Staubli VAL3: TrajJoint.pjx

--- TrajJoint.pjx ---
Parameters version=s7.2.1 stackSize=5000 millimeterUnit=true
Data file=TrajJoint.dtx
Type name=TrajJointItem path=Disk://kernel/template/TrajJointItem/TrajJointItem.pjx

--- TrajJoint.dtx ---
public num nIndexTool
public TrajJointItem tData
  [0]
    jointRx jJoint
    TrajectoryItem tSuper
      [0]
        num distance
        num moveType
        num nTime
        num nStop
        num nTcpAction
        string comment
        bool toStop
        mdesc nom_speed = {tmax=9999}
        InstrItem iInstr[3]
          [0]
            string sType
            string sData
          [1]
            string sType
            string sData
          [2]
            string sType
            string sData
        num nMoveId
public string sID
public num nIndexFrame
